// TwinCAT 3 PLC project PRG_Test_IO
// Company: RafalOS
// ProgramVersion: 3.1.4024.0
// libraries:
//   B_IO, * (RafalOS)
//   Tc2_DataExchange, * (Beckhoff Automation GmbH)
//   Tc2_Standard, * (Beckhoff Automation GmbH)
//   Tc2_System, * (Beckhoff Automation GmbH)
//   Tc3_Module, * (Beckhoff Automation GmbH)
//   TcUnit, * (www.tcunit.org)
// project tree:
//   GVLs/ GVL_Variable.TcGVL
//   / PlcTask.TcTTO
//   POUs/ FB_ButtonTest.TcPOU (not stored), FB_ElectroValveTest.TcPOU (not stored), FB_LampBlinkingTest.TcPOU, FB_SensorTest.TcPOU
//   TESTs/ PRG_Test.TcPOU
// real-time tasks:
//   TASK PlcTask: cycle T#10ms, priority 20, ADS port 350

CONFIGURATION PRG_Test_IO
    RESOURCE PLC ON TwinCAT3
        TASK PlcTask(INTERVAL := T#10ms, PRIORITY := 20);
        PROGRAM PRG_Test WITH PlcTask : PRG_Test;
    END_RESOURCE
END_CONFIGURATION

// ---- GVLs/GVL_Variable.TcGVL
{attribute 'qualified_only'}
VAR_GLOBAL
	fbSaveDataByADS		: Tc2_DataExchange.FB_WriteAdsSymByName;
	bValueToSave		: BOOL;
	bSaved				: BOOL;
	bSave				: BOOL;
	sData				: STRING;

//Czujników	
	senNC				: FB_Sensor_NC;
	senNO				: FB_Sensor_NO;
	sen2NO				: FB_Sensor_NO_2InRow;
//TEST Elektrozawor
	ev3on2_NC			: FB_Electrovalve_3on2_NC;
	ev3on2_NO			: FB_Electrovalve_3on2_NO;
	ev5on2_1C			: FB_Electrovalve_5on2_1Coil;
	ev5on2_2C			: FB_Electrovalve_5on2_2Coil;
	ev5on3_2C_ven		: FB_Electrovalve_5on3_2Coil_Vented;
	ev5on3_2C_inf		: FB_Electrovalve_5on3_2Coil_Infected;
//
	fbLampBlinking		: FB_LampBlinking;
//
	fbButton_NC				: FB_Button_NC;
	fbButton_NO				: FB_Button_NO;

END_VAR

// ---- TESTs/PRG_Test.TcPOU
PROGRAM PRG_Test
VAR
	fbSensorTest			: FB_SensorTest;
	fbElectrovalveTest		: FB_ElectroValveTest;
	fbButtontest			: FB_ButtonTest;
	fbLapmBlinkingTest		: FB_LampBlinkingTest;
END_VAR


	TcUnit.RUN_IN_SEQUENCE ();


GVL_Variable.fbSaveDataByADS (
	bWrite		:= GVL_Variable.bSave,
	sNetId		:= ,
	nPort		:= ,
	sVarName	:= GVL_Variable.sData,
	nSrcAddr	:= ADR (GVL_Variable.bValueToSave),
	nLen		:= SIZEOF (GVL_Variable.bValueToSave),
	tTimeout	:= ,
	eComMode	:= ,
	bBusy		=> GVL_Variable.bSaved,
	bError		=> ,
	nErrorId	=>
);

END_PROGRAM

// ---- POUs/FB_SensorTest.TcPOU
FUNCTION_BLOCK INTERNAL FB_SensorTest EXTENDS TcUnit.FB_TestSuite
VAR
	
END_VAR


T01_TestCzujnikNC ();
T02_TestCzujnikNO ();
T03_TestCzujnikNO_Szereg ();

METHOD PROTECTED T01_TestCzujnikNC
VAR_INST
	iStep			: INT;
END_VAR
IF (TcUnit.TEST_ORDERED ('T01_TestCzujnikNC')) THEN
	CASE iStep OF
	0	:
		GVL_Variable.bValueToSave	:= TRUE;
		GVL_Variable.sData			:= 'GVL_Variable.senNC.bContact';
		GVL_Variable.bSave			:= TRUE;
		iStep						:= iStep + 10;
	10	:
		IF (NOT GVL_Variable.bSaved) THEN
			GVL_Variable.bSave		:= FALSE;
			AssertFalse (Condition := GVL_Variable.senNC.IsActive (), Message := 'K10 - T01 bledny stan');
			iStep					:= iStep + 10;
		END_IF
	20	:
		GVL_Variable.bValueToSave	:= FALSE;
		GVL_Variable.sData			:= 'GVL_Variable.senNC.bContact';
		GVL_Variable.bSave				:= TRUE;
		iStep			:= iStep + 10;
	30	:
		IF (NOT GVL_Variable.bSaved) THEN
			GVL_Variable.bSave			:= FALSE;
			AssertTrue (Condition := GVL_Variable.senNC.IsActive (), Message := 'K20 - T01 bledny stan');
			iStep		:= iStep + 10;
		END_IF
	40	:
		GVL_Variable.bValueToSave	:= TRUE;
		GVL_Variable.sData			:= 'GVL_Variable.senNC.bContact';
		GVL_Variable.bSave				:= TRUE;
		iStep			:= iStep + 10;
	50	:
		IF (NOT GVL_Variable.bSaved) THEN
			GVL_Variable.bSave			:= FALSE;
			AssertFalse (Condition := GVL_Variable.senNC.IsActive (), Message := 'K30 - T01 bledny stan');
			iStep		:= iStep + 10;
		END_IF
	60	:
		iStep			:= 0;
		TcUnit.TEST_FINISHED ();
	END_CASE
END_IF
END_METHOD

METHOD PROTECTED T02_TestCzujnikNO
VAR_INST
	iStep			: INT;
END_VAR
IF (TcUnit.TEST_ORDERED ('T02_TestCzujnikNO')) THEN
	CASE iStep OF
	0	:
		GVL_Variable.bValueToSave	:= FALSE;
		GVL_Variable.sData			:= 'GVL_Variable.senNO.bContact';
		GVL_Variable.bSave			:= TRUE;
		iStep						:= iStep + 10;
	10	:
		IF (NOT GVL_Variable.bSaved) THEN
			GVL_Variable.bSave		:= FALSE;
(*	*)		AssertFalse (Condition := GVL_Variable.senNO.IsActive (), Message := 'K10 - T01 bledny stan');
			iStep					:= iStep + 10;
		END_IF
	20	:
		GVL_Variable.bValueToSave	:= TRUE;
		GVL_Variable.sData			:= 'GVL_Variable.senNO.bContact';
		GVL_Variable.bSave			:= TRUE;
		iStep						:= iStep + 10;
	30	:
		IF (NOT GVL_Variable.bSaved) THEN
			GVL_Variable.bSave		:= FALSE;
(*	*)		AssertTrue (Condition := GVL_Variable.senNO.IsActive (), Message := 'K20 - T01 bledny stan');
			iStep					:= iStep + 10;
		END_IF
	40	:
		GVL_Variable.bValueToSave	:= FALSE;
		GVL_Variable.sData			:= 'GVL_Variable.senNO.bContact';
		GVL_Variable.bSave			:= TRUE;
		iStep						:= iStep + 10;
	50	:
		IF (NOT GVL_Variable.bSaved) THEN
			GVL_Variable.bSave		:= FALSE;
(*	*)		AssertFalse (Condition := GVL_Variable.senNO.IsActive (), Message := 'K30 - T01 bledny stan');
			iStep					:= iStep + 10;
		END_IF
	60	:
		iStep						:= 0;
		TcUnit.TEST_FINISHED ();
	END_CASE	
END_IF
END_METHOD

METHOD PROTECTED T03_TestCzujnikNO_Szereg
VAR_INST
	iStep			: INT;
END_VAR
IF (TcUnit.TEST_ORDERED ('T03_TestCzujnikNO_Szereg')) THEN
	CASE iStep OF
	0	:
		GVL_Variable.bValueToSave	:= FALSE;
		GVL_Variable.sData			:= 'GVL_Variable.sen2NO.bContact';
		GVL_Variable.bSave			:= TRUE;
		iStep						:= iStep + 10;
	10	:
		IF (NOT GVL_Variable.bSaved) THEN
			GVL_Variable.bSave		:= FALSE;
			iStep					:= iStep + 10;
		END_IF
	20	:
		GVL_Variable.bValueToSave	:= FALSE;
		GVL_Variable.sData			:= 'GVL_Variable.sen2NO.bContact2';
		GVL_Variable.bSave			:= TRUE;
		iStep						:= iStep + 10;
	30	:
		IF (NOT GVL_Variable.bSaved) THEN
			GVL_Variable.bSave		:= FALSE;
(*	*)		AssertFalse (Condition := GVL_Variable.sen2NO.IsActive (), Message := 'K30 - T01 bledny stan');
			iStep					:= iStep + 10;
		END_IF
	40	:
		GVL_Variable.bValueToSave	:= TRUE;
		GVL_Variable.sData			:= 'GVL_Variable.sen2NO.bContact';
		GVL_Variable.bSave			:= TRUE;
		iStep						:= iStep + 10;
	50	:
		IF (NOT GVL_Variable.bSaved) THEN
			GVL_Variable.bSave		:= FALSE;
(*	*)		AssertFalse (Condition := GVL_Variable.sen2NO.IsActive (), Message := 'K50 - T01 bledny stan');
			iStep					:= iStep + 10;
		END_IF
	60	:
		GVL_Variable.bValueToSave	:= TRUE;
		GVL_Variable.sData			:= 'GVL_Variable.sen2NO.bContact2';
		GVL_Variable.bSave			:= TRUE;
		iStep						:= iStep + 10;
	70	:
		IF (NOT GVL_Variable.bSaved) THEN
			GVL_Variable.bSave		:= FALSE;
(*	*)		AssertTrue (Condition := GVL_Variable.sen2NO.IsActive (), Message := 'K70 - T01 bledny stan');
			iStep					:= iStep + 10;
		END_IF
	80	:
		GVL_Variable.bValueToSave	:= FALSE;
		GVL_Variable.sData			:= 'GVL_Variable.sen2NO.bContact2';
		GVL_Variable.bSave			:= TRUE;
		iStep						:= iStep + 10;
	90	:
		IF (NOT GVL_Variable.bSaved) THEN
			GVL_Variable.bSave		:= FALSE;
(*	*)		AssertFalse (Condition := GVL_Variable.sen2NO.IsActive (), Message := 'K90 - T01 bledny stan');
			iStep					:= iStep + 10;
		END_IF
	100	:
		GVL_Variable.bValueToSave	:= FALSE;
		GVL_Variable.sData			:= 'GVL_Variable.sen2NO.bContact';
		GVL_Variable.bSave			:= TRUE;
		iStep						:= iStep + 10;
	110	:
		IF (NOT GVL_Variable.bSaved) THEN
			GVL_Variable.bSave		:= FALSE;
(*	*)		AssertFalse (Condition := GVL_Variable.sen2NO.IsActive (), Message := 'K110 - T01 bledny stan');
			iStep					:= 0;
			TcUnit.TEST_FINISHED ();
		END_IF
	END_CASE	
END_IF
END_METHOD

END_FUNCTION_BLOCK

// ---- POUs/FB_LampBlinkingTest.TcPOU
FUNCTION_BLOCK FB_LampBlinkingTest EXTENDS TcUnit.FB_TestSuite
VAR
END_VAR


//T99_test ();

METHOD PRIVATE T99_test
VAR_INST
	bJest		: BOOL;
	bKoniec		: BOOL;
END_VAR
IF (TcUnit.TEST_ORDERED ('T99_Test')) THEN
	IF (NOT bJest) THEN
		bJest					:= TRUE;
		GVL_Variable.fbLampBlinking.SetTimeOn (rIN := 100);
		GVL_Variable.fbLampBlinking.SetTimeOff (rIN := 500);
	END_IF
	GVL_Variable.fbLampBlinking.ExecuteEveryCycle_Test ();
	GVL_Variable.fbLampBlinking.ExecuteEveryCycle_Operation ();
	GVL_Variable.fbLampBlinking.ExecuteEveryCycle_Status ();
	GVL_Variable.fbLampBlinking.ExecuteEveryCycle_Error ();
	IF (bKoniec) THEN
		bJest					:= FALSE;
		TcUnit.TEST_FINISHED ();
	END_IF
END_IF
END_METHOD

END_FUNCTION_BLOCK
